% RSLogix 500 project SMKHOUS.RSS, saved by version 9.05.01.00 %
PROJECT "SMKHOUS"    % processor: MicroLogix 1500 %

PROGRAM FILES
  LAD 2   14 rungs

DATA FILES
  O0 OUTPUT  5 elements
  I1 INPUT  13 elements
  S2 STATUS  66 elements
  B3 BINARY  31 elements
  T4 TIMER  3 elements
  C5 COUNTER  1 elements
  R6 CONTROL  1 elements
  N7 INTEGER  31 elements
  F8 FLOAT  1 elements
  PD9   1 elements

LADDER 2
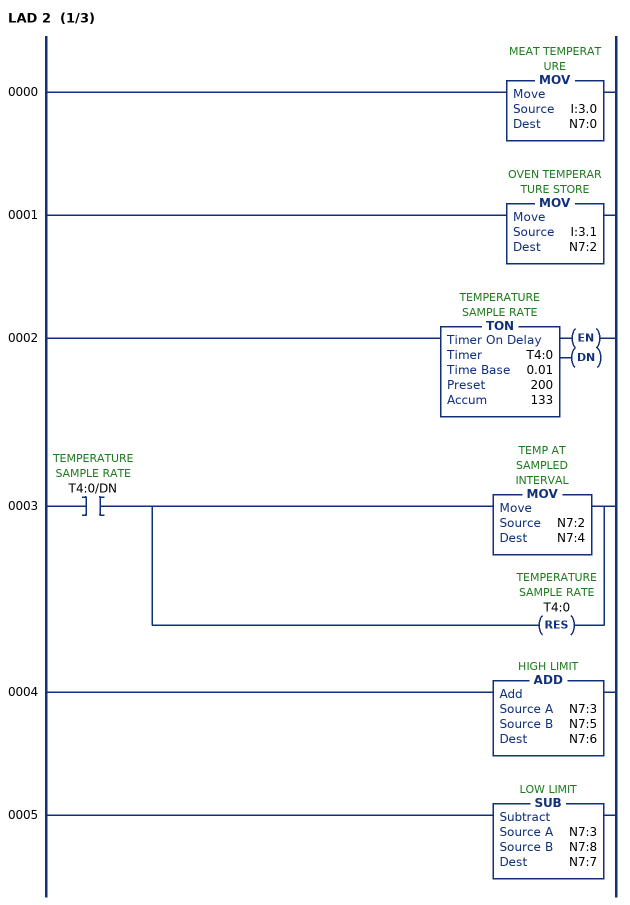
% Rung: 0 %
SOR MOV I:3.0 N7:0 EOR
%   I:3.0  I %
%   N7:0  "MEAT TEMPERATURE" %
% Rung: 1 %
SOR MOV I:3.1 N7:2 EOR
%   N7:2  "OVEN TEMPERARTURE STORE" %
% Rung: 2 %
SOR TON T4:0 0.01 200 133 EOR
%   T4:0  "TEMPERATURE SAMPLE RATE" %
% Rung: 3 %
SOR XIC T4:0/DN BST MOV N7:2 N7:4 NXB RES T4:0 BND EOR
%   T4:0  "TEMPERATURE SAMPLE RATE" %
%   N7:2  "OVEN TEMPERARTURE STORE" %
%   N7:4  "TEMP AT SAMPLED INTERVAL" %
% Rung: 4 %
SOR ADD N7:3 N7:5 N7:6 EOR
%   N7:3  "TEMPERATURE SET POINT" %
%   N7:5  "HIGH DEADBAND" %
%   N7:6  "HIGH LIMIT" %
% Rung: 5 %
SOR SUB N7:3 N7:8 N7:7 EOR
%   N7:3  "TEMPERATURE SET POINT" %
%   N7:8  "LOW DEADBAND" %
%   N7:7  "LOW LIMIT" %

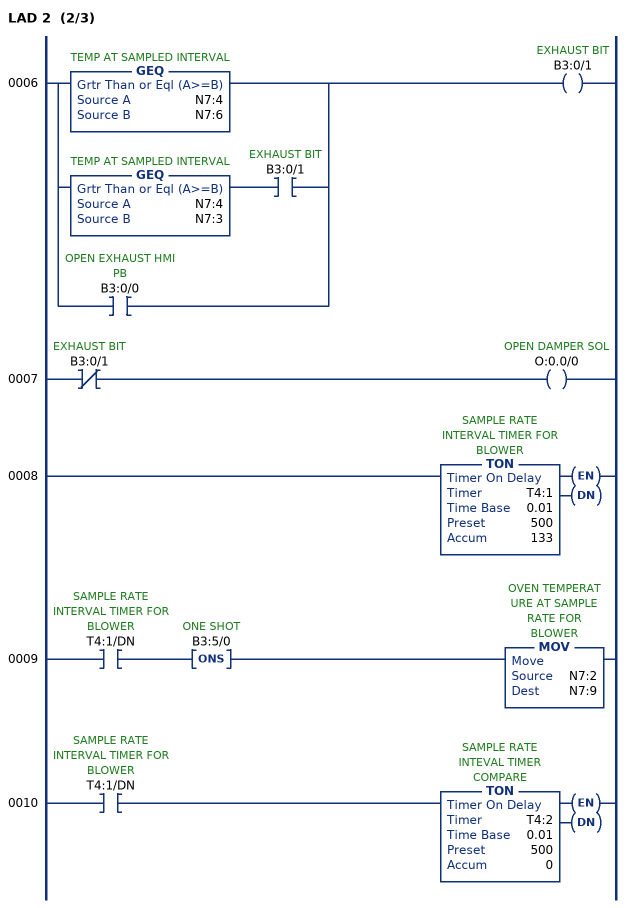
% Rung: 6 %
SOR BST GEQ N7:4 N7:6 NXB GEQ N7:4 N7:3 XIC B3:0/1 NXB XIC B3:0/0 BND OTE B3:0/1 EOR
%   N7:4  "TEMP AT SAMPLED INTERVAL" %
%   N7:6  "HIGH LIMIT" %
%   N7:3  "TEMPERATURE SET POINT" %
%   B3:0/1  "EXHAUST BIT" %
%   B3:0/0  "OPEN EXHAUST HMI PB" %
% Rung: 7 %
SOR XIO B3:0/1 OTE O:0.0/0 EOR
%   B3:0/1  "EXHAUST BIT" %
%   O:0.0/0  "OPEN DAMPER SOL" %
% Rung: 8 %
SOR TON T4:1 0.01 500 133 EOR
%   T4:1  "SAMPLE RATE INTERVAL TIMER FOR BLOWER" %
% Rung: 9 %
SOR XIC T4:1/DN ONS B3:5/0 MOV N7:2 N7:9 EOR
%   T4:1  "SAMPLE RATE INTERVAL TIMER FOR BLOWER" %
%   B3:5/0  "ONE SHOT" %
%   N7:2  "OVEN TEMPERARTURE STORE" %
%   N7:9  "OVEN TEMPERATURE AT SAMPLE RATE FOR BLOWER" %
% Rung: 10 %
SOR XIC T4:1/DN TON T4:2 0.01 500 0 EOR
%   T4:1  "SAMPLE RATE INTERVAL TIMER FOR BLOWER" %
%   T4:2  "SAMPLE RATE INTEVAL TIMER COMPARE" %

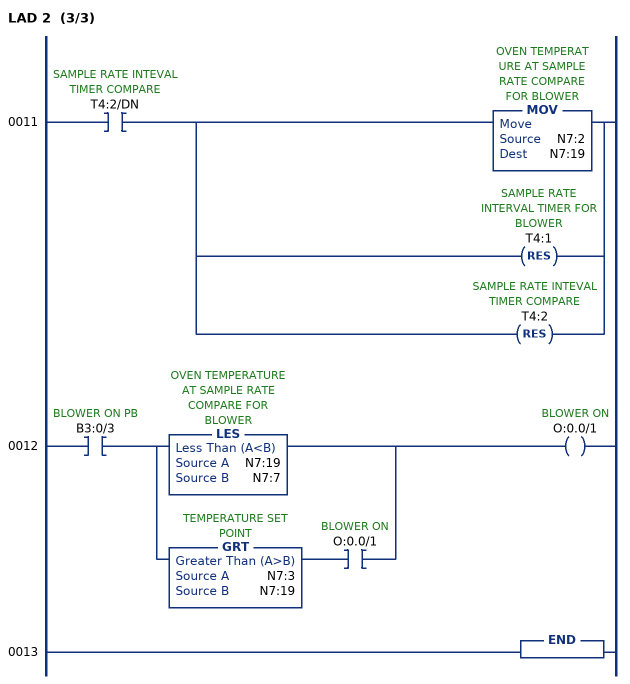
% Rung: 11 %
SOR XIC T4:2/DN BST MOV N7:2 N7:19 NXB RES T4:1 NXB RES T4:2 BND EOR
%   T4:2  "SAMPLE RATE INTEVAL TIMER COMPARE" %
%   N7:2  "OVEN TEMPERARTURE STORE" %
%   N7:19  "OVEN TEMPERATURE AT SAMPLE RATE COMPARE FOR BLOWER" %
%   T4:1  "SAMPLE RATE INTERVAL TIMER FOR BLOWER" %
% Rung: 12 %
SOR XIC B3:0/3 BST LES N7:19 N7:7 NXB GRT N7:3 N7:19 XIC O:0.0/1 BND OTE O:0.0/1 EOR
%   B3:0/3  "BLOWER ON PB" %
%   N7:19  "OVEN TEMPERATURE AT SAMPLE RATE COMPARE FOR BLOWER" %
%   N7:7  "LOW LIMIT" %
%   N7:3  "TEMPERATURE SET POINT" %
%   O:0.0/1  "BLOWER ON" %
% Rung: 13 %
SOR END EOR

OTHER DOCUMENTED ADDRESSES
  B3:0/2  "MEAT GRAPH DECREMENT"
  B3:30/0  "ONE SHOT"
  B3:30/1  "ONE SHOT"
  N7:1  "HOUSE TEMP SETPOINT"
  N7:10  "MEAT GRAPH LOW LIMIT"
  N7:11  "MEAT GRAPH HIGH LIMIT"
  N7:20  "INCREMENT / DECREMENT REGISTER"
  PD9:0  "TEMP PID"

DATA TABLE (non-zero values as saved)
DATA B3
% B3:0 % 0X0008 0X0000 0X0000 0X0000 0X0000 0X0000 0X0000 0X0000 0X0000 0X0000
DATA T4
% .PRE .ACC %
% T4:0 % 200 133
% T4:1 % 500 133
% T4:2 % 500 0
DATA N7
% N7:0 % 73 0 83 90 83 10 100 85 5 84
% N7:10 % 708 200 50 300 0 0 0 0 0 83
% N7:20 % 21920 0 0 0 0 0 0 0 0 0
